// TwinCAT 3 PLC project LabExercise
// ProgramVersion: 3.1.4023.0
// libraries:
//   Tc2_NCI, * (Beckhoff Automation GmbH)
//   Tc2_Standard, * (Beckhoff Automation GmbH)
//   Tc2_System, * (Beckhoff Automation GmbH)
//   Tc3_Module, * (Beckhoff Automation GmbH)
//   VisuDialogs, * (System)
// project tree:
//   Comissioning/Function blocks/ FB_ModifyAutomaticControlSettings.TcPOU (not stored)
//   Comissioning/GVLs/ G_Commissioning.TcGVL (not stored)
//   Comissioning/Struct/ ST_AutomaticControlSettings.TcDUT (not stored), ST_ClosedLoopControlSettings.TcDUT (not stored), ST_MotionReferenceGeneratorSettings.TcDUT (not stored), ST_OpenLoopControlSettings.TcDUT (not stored)
//   ControlBox/Interfaces/ I_ControlBox.TcIO (not stored)
//   ControlBox/Function blocks/ FB_ControlBox.TcPOU (not stored), FB_RealControlBox.TcPOU (not stored), FB_VirtualControlBox.TcPOU (not stored)
//   CraneControl/Function blocks/Sub blocks/ FB_ActiveDamping.TcPOU (not stored), FB_Clock.TcPOU (not stored), FB_ClosedLoopControl.TcPOU (not stored), FB_Joystick.TcPOU (not stored), FB_MotionReferenceGenerator_limit.TcPOU (not stored), FB_OpenLoopControl.TcPOU (not stored), FB_ResetIntegralController.TcPOU (not stored), FB_Status.TcPOU (not stored)
//   CraneControl/Enums/ E_Mode.TcDUT (not stored), E_Status.TcDUT (not stored)
//   CraneControl/Function blocks/Main blocks/ FB_AutomaticControl.TcPOU (not stored), FB_ManualControl.TcPOU (not stored)
//   CraneControl/Functions/ F_BarToEng.TcPOU (not stored), F_LminToEng.TcPOU (not stored), F_RadToDeg.TcPOU (not stored)
//   CraneControl/GVLs/ G_Parameters.TcGVL (not stored), G_Work.TcGVL (not stored)
//   CraneControl/Struct/ ST_ActiveDamping.TcDUT (not stored), ST_Parameters.TcDUT (not stored)
//   / GlobalTextList.TcGTLO (not stored), PlcTask.TcTTO (not stored), Simulator.TcTTO (not stored), Visualization Manager.TcVMO (not stored)
//   HMI/ HMI.TcVIS (not stored)
//   HMI/Sub/ CommissioningHMI.TcVIS (not stored), VirtualControlBox.TcVIS (not stored)
//   Inputs/ FB_JoystickInputScaling.TcPOU (not stored), FB_PositionInputScaling.TcPOU (not stored), FB_PressureInputScaling.TcPOU (not stored), G_Inputs.TcGVL (not stored), G_Sensors.TcGVL
//   Inputs/Struct/ ST_AnalogInput.TcDUT (not stored), ST_AnalogInputStatus.TcDUT (not stored)
//   Internship/ c_FB_ControlBlockWithMonito.TcPOU, FB_Filtering.TcPOU (not stored), FB_InitialPos.TcPOU (not stored), FB_InitialPressure.TcPOU, FB_JoystickRef.TcPOU, FB_Joystick_2.TcPOU, FB_RunClock.TcPOU, FB_MotionReference.TcPOU, FB_SineMotionRef.TcPOU, G_Filtered.TcGVL (not stored), G_OPC_UA.TcGVL, G_Parameter.TcGVL, G_ControlInit.TcGVL
//   Outputs/ FB_ValveOutput.TcPOU, G_Outputs.TcGVL (not stored)
//   Outputs/Struct/ ST_pValveDeadBand.TcDUT, ST_ValveOutput.TcDUT (not stored)
//   ControlBox/GVLs/ G_VirtualControlBox.TcGVL (not stored)
//   Programs/ MAIN.TcPOU, P_ControlBlock.TcPOU, P_Commissioning.TcPOU (not stored), P_ControlBox.TcPOU (not stored), P_CraneControl.TcPOU, P_Filtering.TcPOU, P_Inputs.TcPOU, P_IntialPressure.TcPOU, P_Outputs.TcPOU (not stored), P_RunClock.TcPOU, P_Simulator.TcPOU (not stored)
//   Simulator/ FB_CraneSimulator.TcPOU (not stored), G_Simulator.TcGVL (not stored)
// real-time tasks:
//   TASK PlcTask: cycle T#1ms, priority 20, ADS port 350
//   TASK Simulator: cycle T#100us, priority 1, ADS port 351
// I/O:
//   DEVICE Device 5 (EtherCAT), AmsNetId 10.229.3.117.6.1
//     RIO (EK1100) [EK1100 EtherCAT Coupler (2A E-Bus)]
//       DI (EL1008) [EL1008 8Ch. Dig. Input 24V, 3ms]
//       DO (EL2008) [EL2008 8Ch. Dig. Output 24V, 0.5A]
//       AI1 (EL3068) [EL3068 8Ch. Ana. Input 0-10V]
//       AI2 (EL3068) [EL3068 8Ch. Ana. Input 0-10V]
//       AI3 (EL3174) [EL3174 4Ch. Ana. Input +/-10V Diff., +/-20mA SingleEnded, 16 Bit]
//       AO (EL4104) [EL4104 4Ch. Ana. Output 0-10V, 16bit]
//       End Cap (EL9011) [EL9011 End Terminal]
// variable links:
//   LabExercise/LabExercise Instance <-> Device 5 (EtherCAT)/RIO (EK1100)/AI1 (EL3068)
//     PlcTask Inputs/G_Inputs.stCylPos.nValue <-> AI Standard Channel 3/Value
//     PlcTask Inputs/G_Inputs.stCylPos.stStatus <-> AI Standard Channel 3/Status
//     PlcTask Inputs/G_Inputs.stJoyX.nValue <-> AI Standard Channel 1/Value
//     PlcTask Inputs/G_Inputs.stJoyX.stStatus <-> AI Standard Channel 1/Status
//     PlcTask Inputs/G_Inputs.stJoyY.nValue <-> AI Standard Channel 2/Value
//     PlcTask Inputs/G_Inputs.stJoyY.stStatus <-> AI Standard Channel 2/Status
//     PlcTask Inputs/G_Inputs.stSpoolPos.nValue <-> AI Standard Channel 4/Value
//     PlcTask Inputs/G_Inputs.stSpoolPos.stStatus <-> AI Standard Channel 4/Status
//   LabExercise/LabExercise Instance <-> Device 5 (EtherCAT)/RIO (EK1100)/AI2 (EL3068)
//     PlcTask Inputs/G_Inputs.stPressureCompensator.nValue <-> AI Standard Channel 3/Value
//     PlcTask Inputs/G_Inputs.stPressureCompensator.stStatus <-> AI Standard Channel 3/Status
//     PlcTask Inputs/G_Inputs.stPressureLhvSide.nValue <-> AI Standard Channel 5/Value
//     PlcTask Inputs/G_Inputs.stPressureLhvSide.stStatus <-> AI Standard Channel 5/Status
//     PlcTask Inputs/G_Inputs.stPressurePistonSide.nValue <-> AI Standard Channel 4/Value
//     PlcTask Inputs/G_Inputs.stPressurePistonSide.stStatus <-> AI Standard Channel 4/Status
//     PlcTask Inputs/G_Inputs.stPressureReturn.nValue <-> AI Standard Channel 2/Value
//     PlcTask Inputs/G_Inputs.stPressureReturn.stStatus <-> AI Standard Channel 2/Status
//     PlcTask Inputs/G_Inputs.stPressureRodSide.nValue <-> AI Standard Channel 6/Value
//     PlcTask Inputs/G_Inputs.stPressureRodSide.stStatus <-> AI Standard Channel 6/Status
//     PlcTask Inputs/G_Inputs.stPressureSupply.nValue <-> AI Standard Channel 1/Value
//     PlcTask Inputs/G_Inputs.stPressureSupply.stStatus <-> AI Standard Channel 1/Status
//   LabExercise/LabExercise Instance <-> Device 5 (EtherCAT)/RIO (EK1100)/AI3 (EL3174)
//     PlcTask Inputs/G_Inputs.stFlowReturnSide.nValue <-> AI Standard Channel 1/Value
//     PlcTask Inputs/G_Inputs.stFlowReturnSide.stStatus <-> AI Standard Channel 1/Status
//   LabExercise/LabExercise Instance <-> Device 5 (EtherCAT)/RIO (EK1100)/AO (EL4104)
//     PlcTask Outputs/G_Outputs.stValveOutput.nValveOutput <-> AO Output Channel 1/Analog output
//   LabExercise/LabExercise Instance <-> Device 5 (EtherCAT)/RIO (EK1100)/DI (EL1008)
//     PlcTask Inputs/G_Inputs.bAutoModeSelector <-> Channel 1/Input
//     PlcTask Inputs/G_Inputs.bManualModeSelector <-> Channel 2/Input
//     PlcTask Inputs/G_Inputs.bStartButton <-> Channel 3/Input
//     PlcTask Inputs/G_Inputs.bStopButton <-> Channel 4/Input
//   LabExercise/LabExercise Instance <-> Device 5 (EtherCAT)/RIO (EK1100)/DO (EL2008)
//     PlcTask Outputs/G_Outputs.bGreenLight <-> Channel 1/Output
//     PlcTask Outputs/G_Outputs.bRedLight <-> Channel 2/Output
//     PlcTask Outputs/G_Outputs.stValveOutput.bEnable <-> Channel 3/Output

// ---- Outputs/Struct/ST_pValveDeadBand.TcDUT
TYPE ST_pValveDeadBand :
STRUCT
	fPosMax	: LREAL := 29460; // Positive min value [19660..29490]
	fPosMin	: LREAL := 20800; // Positive max value [19660..29490]
	fNegMin : LREAL := 18500; // Negative max value [9830..19660]
	fNegMax	: LREAL := 9830; // Negative min value [9830..19660]
END_STRUCT
END_TYPE

// ---- Inputs/G_Sensors.TcGVL
{attribute 'qualified_only'}
VAR_GLOBAL
	fJoystickY 					: LREAL;
	fPistonPosition 			: LREAL;
	fPressureSupply				: LREAL;
	fPressureReturn 			: LREAL;
	fPressurePistonSide 		: LREAL;
	fPressureLhvSide  			: LREAL;
	fPressureRodSide 			: LREAL;
END_VAR

// ---- Internship/G_OPC_UA.TcGVL
{attribute 'qualified_only'}
VAR_GLOBAL

	// Mesurements for OPC
	fXRef : LREAL ;
	fXDotRef : LREAL;
	fXReal : LREAL ;
	
	PID_OUT : LREAL;
	Error : LREAL;
	
	fPa : LREAL ;
	fPb : LREAL ;
	fPs : LREAL ;
	
	fPaFiltered : LREAL ;
	fPbFiltered : LREAL ;
	fPsFiltered : LREAL ;
	
	fUnfilteredSignal : LREAL ;
	fFilteredSignal : LREAL ;
	
	
	fU : LREAL ;
	
	fTime : LREAL;
	
END_VAR

// ---- Internship/G_Parameter.TcGVL
{attribute 'qualified_only'}
VAR_GLOBAL
	// Motion Referance parameters
	
	fPositionSetpoint_ms : LREAL := 0.3;
	fRampTime_s : LREAL := 1;
	fMaxSpeed : LREAL := 0.1;
	fHoldPositionTime_s : LREAL := 1;
	fTimeBeforeStarting_s : LREAL := 1;
	fStartVelocity : LREAL := 0;
	
	
	// Enables
	bEnablePID : BOOL := FALSE;
	bEnableU : BOOL := FALSE;	
	bMotionSelect : BOOL := FALSE;
	fCycleTime : LREAL := 0.001;
	
	// PID-constants
	Kp : LREAL := 2.0;
	Ki : LREAL := 0.0;
	Kd : LREAL := 0.0;
	
	// Filter constants
	fPressureFilterNum :LREAL := 0.003137;
	fPressureFilterDenz : LREAL := 1.0;
	fPressureFilterDen : LREAL := -0.9969;
	fPressureFilterInit : LREAL := 0;
	
	fSignalFilterNum :LREAL := 0.09516;
	fSignalFilterDenz : LREAL := 1.0;
	fSignalFilterDen : LREAL := -0.9048;
	fSignalFilterInit : LREAL := 0;
	
END_VAR

// ---- Internship/G_ControlInit.TcGVL
VAR_GLOBAL CONSTANT
	SS_INITIALIZE: SINT := 0;
	SS_STEP: SINT := 1;
END_VAR

// ---- Internship/c_FB_ControlBlockWithMonito.TcPOU
FUNCTION_BLOCK c_FB_ControlBlockWithMonito
VAR_INPUT
	ssMethodType: SINT;
	bEnableU: BOOL;
	bEnablePID: BOOL;
	bEnableFF: BOOL;
	bEnableComp: BOOL;
	
	X_real: LREAL;
	X: LREAL;
	X_dot: LREAL;
	
	Kp: LREAL;
	Ki: LREAL;
	Kd: LREAL;
	
	Ps: LREAL;
	Pa: LREAL;
	Pb: LREAL;
	
	u_filtered: LREAL;
END_VAR
VAR_OUTPUT
	U: LREAL;
	PID_OUT: LREAL;
	Error: LREAL;
	u_unfiltered: LREAL;
END_VAR
VAR
	rtb_TSamp: LREAL;
	temp1: LREAL;
	temp2: LREAL;
	c_DiscreteTimeIntegrator_DS: LREAL;
	DiscreteTransferFcn_states: LREAL;
	UD_DSTATE: LREAL;
	u_FF: LREAL;
	Q_Const : LREAL;
END_VAR


Q_Const := G_Parameter.fQConst;

CASE ssMethodType OF
    SS_INITIALIZE: 
        (* SystemInitialize for Atomic SubSystem: '<Root>/FB_ControlBlockWithMonitoring' *)
        (* InitializeConditions for DiscreteTransferFcn: '<S2>/Discrete Transfer Fcn' *)
        DiscreteTransferFcn_states := 0.0;
        (* InitializeConditions for DiscreteIntegrator: '<S2>/Discrete-Time Integrator' *)
        c_DiscreteTimeIntegrator_DS := 0.0;
        (* InitializeConditions for UnitDelay: '<S4>/UD'
         *
         * Block description for '<S4>/UD':
         *  
         *  Store in Global RAM *)
        UD_DSTATE := 0.0;
        (* End of SystemInitialize for SubSystem: '<Root>/FB_ControlBlockWithMonitoring' *)
    SS_STEP: 
        (* Outputs for Atomic SubSystem: '<Root>/FB_ControlBlockWithMonitoring' *)
        (* Sum: '<S1>/Sum1' incorporates:
         *  Outport: '<Root>/Error' *)
        Error := X - X_real;
        (* SampleTimeMath: '<S4>/TSamp' incorporates:
         *  DiscreteTransferFcn: '<S2>/Discrete Transfer Fcn'
         *
         * About '<S4>/TSamp':
         *  y = u * K where K = 1 / ( w * Ts )
         *   *)
        rtb_TSamp := (0.0009995 * DiscreteTransferFcn_states) * 1000.0;
        (* Switch: '<S1>/Switch' incorporates:
         *  Constant: '<S1>/Constant'
         *  DiscreteIntegrator: '<S2>/Discrete-Time Integrator'
         *  Outport: '<Root>/Error'
         *  Product: '<S2>/Product'
         *  Product: '<S2>/Product1'
         *  Product: '<S2>/Product2'
         *  Sum: '<S2>/Sum1'
         *  Sum: '<S4>/Diff'
         *  UnitDelay: '<S4>/UD'
         *
         * Block description for '<S4>/Diff':
         *  
         *  Add in CPU
         *
         * Block description for '<S4>/UD':
         *  
         *  Store in Global RAM *)

        IF bEnablePID THEN 
            U := ((Kp * Error) + (Ki * c_DiscreteTimeIntegrator_DS)) + ((rtb_TSamp - UD_DSTATE) * Kd);
        ELSE 
            U := 0.0;
        END_IF;
		
		IF bEnableFF THEN 
            u_FF := u_filtered;
        ELSE 
          	u_FF := 0.0;
        END_IF;

        (* End of Switch: '<S1>/Switch' *)
        

        (* Saturate: '<S1>/Saturation1' *)

        IF U > 1.0 THEN 
            PID_OUT := 1.0;
        ELSIF U >= -1.0 THEN 
            PID_OUT := U;
        ELSE 
            PID_OUT := -1.0;
        END_IF;

        (* End of Saturate: '<S1>/Saturation1' *)
        

        (* Switch: '<S1>/Switch1' incorporates:
         *  Constant: '<S1>/Constant1'
         *  Sum: '<S1>/Sum' *)

        IF bEnableU THEN 
            U := u_FF + PID_OUT;
        ELSE 
            U := 0.0;
        END_IF;

        (* End of Switch: '<S1>/Switch1' *)
        

        (* Saturate: '<S1>/Saturation' *)

        IF U > 1.0 THEN 
            (* Outport: '<Root>/U' *)
            U := 1.0;
        ELSIF U < -1.0 THEN 
            (* Outport: '<Root>/U' *)
            U := -1.0;
        END_IF;

        (* End of Saturate: '<S1>/Saturation' *)
        

        (* MATLAB Function: '<S1>/V2Q2u' *)
        (* MATLAB Function 'FB_ControlBlockWithMonitoring/V2Q2u': '<S3>:1' *)
        (* '<S3>:1:3' phi = 0.7130; *)
        (* '<S3>:1:4' A = 33.1/100^2; *)
        (* Area *)
        (* '<S3>:1:5' BW = 0; *)
        (* deadband *)
        (* '<S3>:1:6' SpoolTravel = 7; *)
        (* Maximum Spool Travel *)
        (* '<S3>:1:7' a = (SpoolTravel-BW)/25; *)
        (* Valve Slope Characteristic [mm/(L/min)] *)
        (* '<S3>:1:8' dP_0 = 7e5; *)
        (* Pressure drop with compansator *)
        (* '<S3>:1:10' if x_dot > 0 *)
		
        IF X_dot > 0.0 THEN 
            (* '<S3>:1:11' Q = x_dot * A; *)
            (* Wanted Flow *)
            (* '<S3>:1:12' dP = (Ps-Pa)*1e5; *)
            (* '<S3>:1:13' dp_ref = abs(dP_0/dP); *)
            (* dp_ref = 1; *)
            (* '<S3>:1:15' Q_star = (Q * sqrt(dp_ref)) * 6e4; *)
            (* Referance Flow [L/min] *)
            (* '<S3>:1:16' u = (Q_star * a + BW)/SpoolTravel; *)
			IF NOT(bEnableComp) THEN
            	temp2 := ABS(700000.0 / ((Ps - Pa) * 100000.0));
			ELSE
				temp2 := 1;
			END_IF
			
            u_Unfiltered := (((SQRT(temp2) * (X_dot * 0.00331)) * 60000.0) * (7/Q_Const)) / 7.0;
            (* Control Signal [-1, 1] *)
        ELSIF X_dot < 0.0 THEN 
            (* '<S3>:1:18' elseif x_dot < 0 *)
            (* '<S3>:1:19' Q = x_dot * (A*phi); *)
            (* Wanted Flow *)
            (* '<S3>:1:20' dP = (Ps-Pb)*1e5; *)
            (* '<S3>:1:21' dp_ref = abs(dP_0/dP); *)
            (* dp_ref = 1; *)
            (* '<S3>:1:23' Q_star = (Q * sqrt(dp_ref)) * 6e4; *)
            (* Referance Flow [L/min] *)
            (* '<S3>:1:24' u = (Q_star * a - BW)/SpoolTravel; *)
			IF NOT(bEnableComp) THEN
            	temp1 := ABS(700000.0 / ((Ps - Pb) * 100000.0));
			ELSE
				temp1 := 1;
			END_IF
            u_Unfiltered := (((SQRT(temp1) * (X_dot * 0.00236003)) * 60000.0) * (7/Q_Const)) / 7.0;
            (* Control Signal [-1, 1] *)
        ELSE 
            (* '<S3>:1:26' else *)
            (* '<S3>:1:27' u = 0; *)
            u_Unfiltered := 0.0;
        END_IF;

        (* End of MATLAB Function: '<S1>/V2Q2u' *)
        

        (* Saturate: '<S1>/Saturation2' *)

        IF u_Unfiltered > 1.0 THEN 
            (* Outport: '<Root>/u_Unfiltered' *)
            u_Unfiltered := 1.0;
        ELSIF u_Unfiltered < -1.0 THEN 
            (* Outport: '<Root>/u_Unfiltered' *)
            u_Unfiltered := -1.0;
        END_IF;

        (* End of Saturate: '<S1>/Saturation2' *)
        

        (* Update for DiscreteTransferFcn: '<S2>/Discrete Transfer Fcn' incorporates:
         *  Outport: '<Root>/Error' *)
        DiscreteTransferFcn_states := Error - (-0.999 * DiscreteTransferFcn_states);
        (* u_ffpdate for DiscreteIntegrator: '<S2>/Discrete-Time Integrator' incorporates:
         *  Ou_fftport: '<Root>/Error' *)
        c_DiscreteTimeIntegrator_DS := (0.001 * Error) + c_DiscreteTimeIntegrator_DS;
        (* u_ffpdate for u_ffnitDelay: '<S4>/u_ffD'
         *
         * Block description for '<S4>/u_ffD':
         *  
         *  Store in Global RAM *)
        UD_DSTATE := rtb_TSamp;
        (* End of Ou_fftpu_ffts for Su_ffbSystem: '<Root>/FB_ControlBlockWithMonitoring' *)
END_CASE;

END_FUNCTION_BLOCK

// ---- Internship/FB_InitialPressure.TcPOU
FUNCTION_BLOCK FB_InitialPressure
VAR_INPUT
	bEnable : BOOL;
	fCurrentPressure : LREAL;
END_VAR
VAR_OUTPUT
	fInitialPressure : LREAL;
END_VAR
VAR
END_VAR

IF bEnable THEN
	fInitialPressure := fInitialPressure;
ELSE 
	fInitialPressure := fCurrentPressure;
END_IF

END_FUNCTION_BLOCK

// ---- Internship/FB_JoystickRef.TcPOU
FUNCTION_BLOCK FB_JoystickRef
VAR_INPUT
	ssMethodType: SINT;
	Joystick: LREAL;
	XRealRef: LREAL;
END_VAR
VAR_OUTPUT
	fPositionReferance_m: LREAL;
	fVelocityReferance_ms: LREAL;
END_VAR
VAR
	c_DiscreteTimeIntegrator_IC: USINT;
	c_DiscreteTimeIntegrator_DS: LREAL;
END_VAR



CASE ssMethodType OF
    SS_INITIALIZE: 
        (* SystemInitialize for Atomic SubSystem: '<Root>/FB_Joystick' *)
        (* InitializeConditions for DiscreteIntegrator: '<S1>/Discrete-Time Integrator' *)
        c_DiscreteTimeIntegrator_IC := 1;
        (* End of SystemInitialize for SubSystem: '<Root>/FB_Joystick' *)
    SS_STEP: 
        (* Outputs for Atomic SubSystem: '<Root>/FB_Joystick' *)
        (* Gain: '<S1>/Gain' *)
        fVelocityReferance_ms := G_Parameter.fMaxSpeed * Joystick;
        (* DiscreteIntegrator: '<S1>/Discrete-Time Integrator' *)

        IF c_DiscreteTimeIntegrator_IC <> 0 THEN 
            c_DiscreteTimeIntegrator_DS := XRealRef;

            IF c_DiscreteTimeIntegrator_DS > 0.45 THEN 
                c_DiscreteTimeIntegrator_DS := 0.45;
            ELSIF c_DiscreteTimeIntegrator_DS < 0.0 THEN 
                c_DiscreteTimeIntegrator_DS := 0.0;
            END_IF;

        END_IF;

        (* Outport: '<Root>/fPositionReferance_m' incorporates:
         *  DiscreteIntegrator: '<S1>/Discrete-Time Integrator' *)
        fPositionReferance_m := c_DiscreteTimeIntegrator_DS;
        (* Update for DiscreteIntegrator: '<S1>/Discrete-Time Integrator' *)
        c_DiscreteTimeIntegrator_IC := 0;
        c_DiscreteTimeIntegrator_DS := (0.2 * fVelocityReferance_ms) + c_DiscreteTimeIntegrator_DS;

        IF c_DiscreteTimeIntegrator_DS > 0.45 THEN 
            c_DiscreteTimeIntegrator_DS := 0.45;
        ELSIF c_DiscreteTimeIntegrator_DS < 0.0 THEN 
            c_DiscreteTimeIntegrator_DS := 0.0;
        END_IF;

        (* End of Update for DiscreteIntegrator: '<S1>/Discrete-Time Integrator' *)
        (* End of Outputs for SubSystem: '<Root>/FB_Joystick' *)
END_CASE;

END_FUNCTION_BLOCK

// ---- Internship/FB_Joystick_2.TcPOU
FUNCTION_BLOCK FB_Joystick_2
VAR_INPUT
	ssMethodType: SINT;
	Joystick: LREAL;
	XInital: LREAL;
END_VAR
VAR_OUTPUT
	fPositionReferance_m: LREAL;
	fVelocityReferance_ms: LREAL;
END_VAR
VAR
	c_DiscreteTimeIntegrator_IC: USINT;
	c_DiscreteTimeIntegrator_DS: LREAL;
END_VAR



CASE ssMethodType OF
    SS_INITIALIZE: 
        (* SystemInitialize for Atomic SubSystem: '<Root>/FB_Joystick' *)
        (* InitializeConditions for DiscreteIntegrator: '<S1>/Discrete-Time Integrator' *)
        c_DiscreteTimeIntegrator_IC := 1;
        (* End of SystemInitialize for SubSystem: '<Root>/FB_Joystick' *)
    SS_STEP: 
        (* Outputs for Atomic SubSystem: '<Root>/FB_Joystick' *)
        (* Gain: '<S1>/Gain' *)
        fVelocityReferance_ms := G_Parameter.fMaxSpeed * Joystick;
        (* DiscreteIntegrator: '<S1>/Discrete-Time Integrator' *)

        IF c_DiscreteTimeIntegrator_IC <> 0 THEN 
            c_DiscreteTimeIntegrator_DS := XInital;

            IF c_DiscreteTimeIntegrator_DS > 0.45 THEN 
                c_DiscreteTimeIntegrator_DS := 0.45;
            ELSIF c_DiscreteTimeIntegrator_DS < 0.0 THEN 
                c_DiscreteTimeIntegrator_DS := 0.0;
            END_IF;

        END_IF;

        (* Outport: '<Root>/fPositionReferance_m' incorporates:
         *  DiscreteIntegrator: '<S1>/Discrete-Time Integrator' *)
        fPositionReferance_m := c_DiscreteTimeIntegrator_DS;
        (* Update for DiscreteIntegrator: '<S1>/Discrete-Time Integrator' *)
        c_DiscreteTimeIntegrator_IC := 0;
        c_DiscreteTimeIntegrator_DS := (0.001 * fVelocityReferance_ms) + c_DiscreteTimeIntegrator_DS;

        IF c_DiscreteTimeIntegrator_DS > 0.45 THEN 
            c_DiscreteTimeIntegrator_DS := 0.45;
        ELSIF c_DiscreteTimeIntegrator_DS < 0.0 THEN 
            c_DiscreteTimeIntegrator_DS := 0.0;
        END_IF;

        (* End of Update for DiscreteIntegrator: '<S1>/Discrete-Time Integrator' *)
        (* End of Outputs for SubSystem: '<Root>/FB_Joystick' *)
END_CASE;

END_FUNCTION_BLOCK

// ---- Internship/FB_RunClock.TcPOU
FUNCTION_BLOCK FB_RunClock
VAR_INPUT
	bStart 		: BOOL;
	bStop 		: BOOL;
	fCycleTime  : LREAL;
END_VAR
VAR_OUTPUT
	fTime : LREAL;
END_VAR
VAR
	bOnOff : BOOL;
END_VAR

IF bStop OR (G_Work.eStatus = E_Status.Off) THEN
	bOnOff := FALSE;
	fTime := 0.0;
ELSIF bOnOff OR bStart AND (G_Work.eStatus = E_Status.Starting) THEN
	bOnOff := TRUE;
	fTime := fTime + fCycleTime;
END_IF

END_FUNCTION_BLOCK

// ---- Internship/FB_MotionReference.TcPOU
FUNCTION_BLOCK FB_MotionReference
VAR_INPUT
	fStartPosition_m: LREAL;
	fStartVelocity_m: LREAL;
	fPositionSetpoint_ms: LREAL;
	fVelocitySetpoint_m: LREAL;
	fTimeBeforeStarting_s: LREAL;
	fRampTime_s: LREAL;
	fHoldPositionTime_s: LREAL;
	fClock_s: LREAL;
	bEnable: BOOL;
END_VAR
VAR_OUTPUT
	fPositionReference_m: LREAL;
	fVelocityReference_ms: LREAL;
END_VAR
VAR
	Error: DINT;
	slopeExt: LREAL;
	slopeRetr: LREAL;
	tHold: LREAL;
	x1: LREAL;
	x4: LREAL;
	x1_tmp_tmp: LREAL;
	x4_tmp: LREAL;
	x4_tmp_tmp: LREAL;
	x4_tmp_tmp_0: LREAL;
	x1_tmp: LREAL;
END_VAR


(* Outputs for Atomic SubSystem: '<Root>/FB_MotionReferenceGenerator_nolimit' *)
(* MATLAB Function: '<S1>/WaveSignal' *)
(* MATLAB Function 'FB_MotionReferenceGenerator_nolimit/WaveSignal': '<S2>:1' *)
(* '<S2>:1:2' x_SP = x_ref - x0; *)
(* '<S2>:1:3' vs=v_ref; *)
(* '<S2>:1:4' slopeExt=v0-vs; *)
slopeExt := fStartVelocity_m - fVelocitySetpoint_m;
(* '<S2>:1:5' slopeRetr=-vs-v0; *)
slopeRetr := ( -fVelocitySetpoint_m) - fStartVelocity_m;
(* '<S2>:1:7' as = vs/tRamp; *)
(* '<S2>:1:8' s_acc=(vs^2-v0^2)/as; *)
(* '<S2>:1:10' tHold=(x_SP-s_acc)/vs; *)
tHold := ((fPositionSetpoint_ms - fStartPosition_m) - (((fVelocitySetpoint_m * fVelocitySetpoint_m) - (fStartVelocity_m * fStartVelocity_m)) / (fVelocitySetpoint_m / fRampTime_s))) / fVelocitySetpoint_m;
(* '<S2>:1:12' if tHold < 0 *)

IF tHold < 0.0 THEN 
    (* '<S2>:1:13' Error = 1; *)
    Error := 1;
ELSE 
    (* '<S2>:1:14' else *)
    (* '<S2>:1:15' Error = 0; *)
    Error := 0;
END_IF;

(* '<S2>:1:18' t1=tRamp; *)
(* '<S2>:1:19' t2=tHold; *)
(* '<S2>:1:20' t3=tRamp; *)
(* '<S2>:1:21' t4=tWait; *)
(* '<S2>:1:22' t5=t1; *)
(* '<S2>:1:23' t6=t2; *)
(* '<S2>:1:24' t7=t3; *)
(* '<S2>:1:26' x = x0; *)
(* '<S2>:1:27' x1 = x0 + v0*((t0+t1)-t0)-(slopeExt/t1)*((t0+t1)-t0)^2/2; *)
x1_tmp_tmp := fTimeBeforeStarting_s + fRampTime_s;
x4 := x1_tmp_tmp - fTimeBeforeStarting_s;
x1_tmp := slopeExt / fRampTime_s;
x1 := ((x4 * fStartVelocity_m) + fStartPosition_m) - ((x1_tmp * (x4 * x4)) / 2.0);
(* '<S2>:1:28' x2 = x1 + vs*((t0+t1+t2)-(t0+t1)); *)
(* '<S2>:1:29' x4 = x_ref - v0*((t0+t1+t2+t3+t4+t5)-(t0+t1+t2+t3+t4))+(slopeRetr/t5)*((t0+t1+t2+t3+t4+t5)-(t0+t1+t2+t3+t4))^2/2; *)
x4_tmp_tmp := x1_tmp_tmp + tHold;
x4_tmp_tmp_0 := x4_tmp_tmp + fRampTime_s;
x4_tmp := x4_tmp_tmp_0 + fHoldPositionTime_s;
x4 := (x4_tmp + fRampTime_s) - x4_tmp;
x4 := (fPositionSetpoint_ms - (x4 * fStartVelocity_m)) + (((slopeRetr / fRampTime_s) * (x4 * x4)) / 2.0);
(* '<S2>:1:30' x5 = x4-vs*((t0+t1+t2+t3+t4+t5+t6)-(t0+t1+t2+t3+t4+t5)); *)
(* '<S2>:1:32' if Error == 1 *)

IF Error = 1 THEN 
    (* '<S2>:1:33' x = x0; *)
    fPositionReference_m := fStartPosition_m;
    (* '<S2>:1:34' v = v0; *)
    fVelocityReference_ms := fStartVelocity_m;
ELSIF (fClock_s >= 0.0) AND (fClock_s < fTimeBeforeStarting_s) THEN 
    (* '<S2>:1:35' elseif t>=0 && t<t0 *)
    (* '<S2>:1:36' x = x0; *)
    fPositionReference_m := fStartPosition_m;
    (* '<S2>:1:37' v = v0; *)
    fVelocityReference_ms := fStartVelocity_m;
ELSIF (fClock_s >= fTimeBeforeStarting_s) AND (fClock_s < x1_tmp_tmp) THEN 
    (* '<S2>:1:38' elseif t>=t0 && t<(t0+t1) *)
    (* '<S2>:1:39' x = x0 + v0*(t-t0)-(slopeExt/t1)*(t-t0)^2/2; *)
    slopeExt := fClock_s - fTimeBeforeStarting_s;
    fPositionReference_m := ((slopeExt * fStartVelocity_m) + fStartPosition_m) - ((x1_tmp * (slopeExt * slopeExt)) / 2.0);
    (* '<S2>:1:40' v = v0-(slopeExt/t1)*(t-t0); *)
    fVelocityReference_ms := fStartVelocity_m - (x1_tmp * slopeExt);
ELSIF (fClock_s >= x1_tmp_tmp) AND (fClock_s < x4_tmp_tmp) THEN 
    (* '<S2>:1:41' elseif t>=(t0+t1) && t<(t0+t1+t2) *)
    (* '<S2>:1:42' x = x1 + vs*(t-(t0+t1)); *)
    fPositionReference_m := ((fClock_s - x1_tmp_tmp) * fVelocitySetpoint_m) + x1;
    (* '<S2>:1:43' v = vs; *)
    fVelocityReference_ms := fVelocitySetpoint_m;
ELSIF (fClock_s >= x4_tmp_tmp) AND (fClock_s < x4_tmp_tmp_0) THEN 
    (* '<S2>:1:44' elseif t>=(t0+t1+t2) && t<(t0+t1+t2+t3) *)
    (* '<S2>:1:45' x = x2+vs*(t-(t0+t1+t2))+(slopeExt/t3)*(t-(t0+t1+t2))^2/2; *)
    tHold := (fTimeBeforeStarting_s + fRampTime_s) + tHold;
    slopeRetr := fClock_s - tHold;
    fPositionReference_m := ((((tHold - x1_tmp_tmp) * fVelocitySetpoint_m) + x1) + (slopeRetr * fVelocitySetpoint_m)) + ((x1_tmp * (slopeRetr * slopeRetr)) / 2.0);
    (* '<S2>:1:46' v = vs+(slopeExt/t3)*(t-(t0+t1+t2)); *)
    fVelocityReference_ms := (slopeRetr * (slopeExt / fRampTime_s)) + fVelocitySetpoint_m;
ELSIF (fClock_s >= x4_tmp_tmp_0) AND (fClock_s < x4_tmp) THEN 
    (* '<S2>:1:47' elseif t>=(t0+t1+t2+t3) && t<(t0+t1+t2+t3+t4) *)
    (* '<S2>:1:48' x = x_ref; *)
    fPositionReference_m := fPositionSetpoint_ms;
    (* '<S2>:1:49' v = v0; *)
    fVelocityReference_ms := fStartVelocity_m;
ELSE 
    x1_tmp := ((x1_tmp_tmp + tHold) + fRampTime_s) + fHoldPositionTime_s;
    slopeExt := x1_tmp + fRampTime_s;

    IF (fClock_s >= x1_tmp) AND (fClock_s < slopeExt) THEN 
        (* '<S2>:1:50' elseif t>=(t0+t1+t2+t3+t4) && t<(t0+t1+t2+t3+t4+t5) *)
        (* '<S2>:1:51' x = x_ref - v0*(t-(t0+t1+t2+t3+t4))+(slopeRetr/t5)*(t-(t0+t1+t2+t3+t4))^2/2; *)
        tHold := fClock_s - x1_tmp;
        slopeRetr := slopeRetr / fRampTime_s;
        fPositionReference_m := (fPositionSetpoint_ms - (tHold * fStartVelocity_m)) + ((slopeRetr * (tHold * tHold)) / 2.0);
        (* '<S2>:1:52' v = v0+(slopeRetr/t5)*(t-(t0+t1+t2+t3+t4)); *)
        fVelocityReference_ms := (tHold * slopeRetr) + fStartVelocity_m;
    ELSE 
        x1_tmp := slopeExt + tHold;

        IF (fClock_s >= slopeExt) AND (fClock_s < x1_tmp) THEN 
            (* '<S2>:1:53' elseif t>=(t0+t1+t2+t3+t4+t5) && t<(t0+t1+t2+t3+t4+t5+t6) *)
            (* '<S2>:1:54' x = x4-vs*(t-(t0+t1+t2+t3+t4+t5)); *)
            fPositionReference_m := x4 - ((fClock_s - slopeExt) * fVelocitySetpoint_m);
            (* '<S2>:1:55' v = -vs; *)
            fVelocityReference_ms :=  -fVelocitySetpoint_m;
        ELSIF (fClock_s >= x1_tmp) AND (fClock_s < (x1_tmp + fRampTime_s)) THEN 
            (* '<S2>:1:56' elseif t>=(t0+t1+t2+t3+t4+t5+t6) && t<(t0+t1+t2+t3+t4+t5+t6+t7) *)
            (* '<S2>:1:57' x = x5-vs*(t-(t0+t1+t2+t3+t4+t5+t6))-(slopeRetr/t3)*(t-(t0+t1+t2+t3+t4+t5+t6))^2/2; *)
            tHold := fClock_s - x1_tmp;
            slopeRetr := slopeRetr / fRampTime_s;
            fPositionReference_m := ((x4 - ((x1_tmp - slopeExt) * fVelocitySetpoint_m)) - (tHold * fVelocitySetpoint_m)) - ((slopeRetr * (tHold * tHold)) / 2.0);
            (* '<S2>:1:58' v = -vs-(slopeRetr/t3)*(t-(t0+t1+t2+t3+t4+t5+t6)); *)
            fVelocityReference_ms := ( -fVelocitySetpoint_m) - (tHold * slopeRetr);
        ELSE 
            (* '<S2>:1:59' else *)
            (* '<S2>:1:60' x = x0; *)
            fPositionReference_m := fStartPosition_m;
            (* '<S2>:1:61' v = v0; *)
            fVelocityReference_ms := fStartVelocity_m;
        END_IF;

    END_IF;

END_IF;

(* End of MATLAB Function: '<S1>/WaveSignal' *)


(* Switch: '<S1>/Switch' incorporates:
 *  Switch: '<S1>/Switch1' *)
(* '<S2>:1:64' T = t0+t1+t2+t3+t4+t5+t6+t7; *)

IF  NOT bEnable THEN 
    (* Outport: '<Root>/fVelocityReference_ms' *)
    fVelocityReference_ms := fStartVelocity_m;
    (* Outport: '<Root>/fPositionReference_m' *)
    fPositionReference_m := fStartPosition_m;
END_IF;

(* End of Switch: '<S1>/Switch' *)
(* End of Outputs for SubSystem: '<Root>/FB_MotionReferenceGenerator_nolimit' *)

END_FUNCTION_BLOCK

// ---- Internship/FB_SineMotionRef.TcPOU
FUNCTION_BLOCK FB_SineMotionRef
VAR_INPUT
	ssMethodType: SINT;
	fTime: LREAL;
	fPos_Ramp_Time: LREAL;
	fPeak_pos: LREAL;
	fStart_vel: LREAL;
	fStart_time: LREAL;
	fHold_time: LREAL;
	fXReal: LREAL;
END_VAR
VAR_OUTPUT
	X_dot: LREAL;
	X: LREAL;
END_VAR
VAR
	peak_vel: LREAL;
	amplitude_vel: LREAL;
	c_DiscreteTimeIntegrator_DS: LREAL;
END_VAR



CASE ssMethodType OF
    SS_INITIALIZE: 
        (* SystemInitialize for Atomic SubSystem: '<Root>/FB_SineMotionRef' *)
        (* InitializeConditions for DiscreteIntegrator: '<S1>/Discrete-Time Integrator' *)
        c_DiscreteTimeIntegrator_DS := 0.0;
        (* End of SystemInitialize for SubSystem: '<Root>/FB_SineMotionRef' *)
    SS_STEP: 
        (* Outputs for Atomic SubSystem: '<Root>/FB_SineMotionRef' *)
        (* MATLAB Function: '<S1>/MATLAB Function' *)
        (* MATLAB Function 'FB_SineMotionRef/MATLAB Function': '<S2>:1' *)
        (* '<S2>:1:2' max_pos = peak_pos-start_pos; *)
        (* '<S2>:1:3' peak_vel = max_pos*2/pos_ramp_time; *)
        peak_vel := ((fPeak_pos - fXReal) * 2.0) / fPos_Ramp_Time;
        (* '<S2>:1:4' pos_sat = peak_vel*pos_ramp_time/2 +start_pos; *)
        (* '<S2>:1:5' amplitude_vel = peak_vel/2; *)
        amplitude_vel := peak_vel / 2.0;
        (* '<S2>:1:6' if pos_sat <= 0.4 *)

        IF (((peak_vel * fPos_Ramp_Time) / 2.0) + fXReal) <= 0.4 THEN 
            (* '<S2>:1:7' if time<start_time *)

            IF fTime < fStart_time THEN 
                (* '<S2>:1:8' X_dot=start_vel; *)
                X_dot := fStart_vel;
            ELSIF fTime <= (fPos_Ramp_Time + fStart_time) THEN 
                (* '<S2>:1:9' elseif time<=pos_ramp_time+start_time *)
                (* '<S2>:1:10' X_dot=amplitude_vel-amplitude_vel*cos((2*(time-start_time))/pos_ramp_time*pi)+start_vel; *)
                X_dot := (amplitude_vel - (COS((((fTime - fStart_time) * 2.0) / fPos_Ramp_Time) * 3.1415926535897931) * amplitude_vel)) + fStart_vel;
            ELSIF fTime < ((fHold_time + fPos_Ramp_Time) + fStart_time) THEN 
                (* '<S2>:1:11' elseif time<hold_time+pos_ramp_time+start_time *)
                (* '<S2>:1:12' X_dot=start_vel; *)
                X_dot := fStart_vel;
            ELSIF fTime < (((2.0 * fPos_Ramp_Time) + fHold_time) + fStart_time) THEN 
                (* '<S2>:1:13' elseif time< hold_time+2*pos_ramp_time+start_time *)
                (* '<S2>:1:14' X_dot=-(amplitude_vel-amplitude_vel*cos((2*(time-(start_time +hold_time+pos_ramp_time)))/pos_ramp_time*pi)+start_vel); *)
                X_dot :=  -((amplitude_vel - (COS((((fTime - ((fStart_time + fHold_time) + fPos_Ramp_Time)) * 2.0) / fPos_Ramp_Time) * 3.1415926535897931) * amplitude_vel)) + fStart_vel);
            ELSE 
                (* '<S2>:1:15' else *)
                (* '<S2>:1:16' X_dot=start_vel; *)
                X_dot := fStart_vel;
            END_IF;

        ELSE 
            (* '<S2>:1:18' else *)
            (* '<S2>:1:19' X_dot=0; *)
            X_dot := 0.0;
        END_IF;

        (* End of MATLAB Function: '<S1>/MATLAB Function' *)
        

        (* Outport: '<Root>/X' incorporates:
         *  DiscreteIntegrator: '<S1>/Discrete-Time Integrator'
         *  Sum: '<S1>/Sum' *)
        X := c_DiscreteTimeIntegrator_DS + fXReal;
        (* Update for DiscreteIntegrator: '<S1>/Discrete-Time Integrator' *)
        c_DiscreteTimeIntegrator_DS := (0.001 * X_dot) + c_DiscreteTimeIntegrator_DS;
        (* End of Outputs for SubSystem: '<Root>/FB_SineMotionRef' *)
END_CASE;

END_FUNCTION_BLOCK

// ---- Outputs/FB_ValveOutput.TcPOU
FUNCTION_BLOCK FB_ValveOutput
VAR_INPUT
	bEnable 			: BOOL;
	stParam 			: ST_Parameters;
	fNormalizedInput 	: LREAL;
END_VAR
VAR_OUTPUT
	bEnableValveOutput : BOOL;
	nOutput : INT; 
END_VAR
VAR
	nOffset 	: INT := 19630;
	nMaxValue	: INT := 29460;
	nMinValue 	: INT :=  9830;
	nTempOutput : INT;
END_VAR

IF fNormalizedInput > 0.0 THEN
	nTempOutput := LREAL_TO_INT(ABS(fNormalizedInput*(stParam.stValveDeadBand.fPosMax - stParam.stValveDeadBand.fPosMin) + stParam.stValveDeadBand.fPosMin));
ELSIF fNormalizedInput < 0.0 THEN
	nTempOutput := LREAL_TO_INT(ABS(fNormalizedInput*(stParam.stValveDeadBand.fNegMax - stParam.stValveDeadBand.fNegMin) - stParam.stValveDeadBand.fNegMin));
ELSE
	nTempOutput := nOffset;
END_IF

IF NOT(bEnable) THEN
	nOutput := nOffset;
	bEnableValveOutput := FALSE;
ELSE
	nOutput := LIMIT(nMinValue, nTempOutput, nMaxValue);
	bEnableValveOutput := TRUE; 
END_IF

END_FUNCTION_BLOCK

// ---- Programs/MAIN.TcPOU
PROGRAM MAIN
VAR
END_VAR

P_Commissioning();
P_ControlBox();
P_Filtering();
P_CraneControl();
P_ControlBlock();
P_Outputs();
P_Inputs();
P_RunClock();

END_PROGRAM

// ---- Programs/P_Filtering.TcPOU
PROGRAM P_Filtering
VAR
	fbControlBlock : c_FB_ControlBlockWithMonito;
	fbFilterPa : FB_Filtering;
	fbFilterPb : FB_Filtering;
	fbFilterPs : FB_Filtering;
	fbFilterU : FB_Filtering;
END_VAR

fbFilterPa(
	ssMethodType := 1,
	Signal := G_Sensors.fPressurePistonSide,
	Num := G_Parameter.fPressureFilterNum,
	Denz := G_Parameter.fPressureFilterDenz,
	Den := G_Parameter.fPressureFilterDen,
	Initial := G_Parameter.fPressureFilterInit,
	
	Signal_Filtered => G_Filtered.fPressurePistonSideFiltered,
	Signal_Filtered => G_OPC_UA.fPaFiltered
);

fbFilterPb(
	ssMethodType := 1,
	Signal := G_Sensors.fPressureRodSide,
	Num := G_Parameter.fPressureFilterNum,
	Denz := G_Parameter.fPressureFilterDenz,
	Den := G_Parameter.fPressureFilterDen,
	Initial := G_Parameter.fPressureFilterInit,
	
	Signal_Filtered => G_Filtered.fPressureRodSideFiltered,
	Signal_Filtered => G_OPC_UA.fPbFiltered
);

fbFilterPs(
	ssMethodType := 1,
	Signal := G_Sensors.fPressureSupply,
	Num := G_Parameter.fPressureFilterNum,
	Denz := G_Parameter.fPressureFilterDenz,
	Den := G_Parameter.fPressureFilterDen,
	Initial := G_Parameter.fPressureFilterInit,
	
	Signal_Filtered => G_Filtered.fPressureSupplyFiltered,
	Signal_Filtered => G_OPC_UA.fPsFiltered
);

fbFilterU(
	ssMethodType := 1,
	Signal := G_Filtered.fValveOutputUnfiltered,
	Num := G_Parameter.fSignalFilterNum,
	Denz := G_Parameter.fSignalFilterDenz,
	Den := G_Parameter.fSignalFilterDen,
	Initial := G_Parameter.fSignalFilterInit,
	
	Signal_Filtered => G_Filtered.fValveOutputFiltered,
	Signal_Filtered => G_OPC_UA.fFilteredSignal
);

END_PROGRAM

// ---- Programs/P_CraneControl.TcPOU
PROGRAM P_CraneControl
VAR
 	fbStatus 					: FB_Status;
	fbRunningClock 				: FB_Clock;
	fbManualControl 			: FB_ManualControl; 
	bEnableManualControl 		: BOOL;
	fbAutomaticControl 			: FB_AutomaticControl;
	bEnableAutomaticControl 	: BOOL; 
	fbActiveDamping 			: FB_ActiveDamping;
	fControlOutputNormalized 	: LREAL; 
	
	ADtest0 : LREAL;
	ADtest1 : LREAL;
	ADtest2 : LREAL;
	ADtest : BOOL;
END_VAR

fbStatus(
bFault := G_Work.bFault,
eMode := G_Work.eMode,
fTime := fbRunningClock.fTime,
eStatus => G_Work.eStatus
);

fbRunningClock(
	bStart := (fbStatus.eStatus = E_Status.Starting) OR (fbStatus.eStatus = E_Status.Running),
	bStop := (fbStatus.eStatus = E_Status.Stopping),
	fCycleTime := G_Parameters.stParam.fCyclicTime
);


fbManualControl(
	eMode := G_Work.eMode,
	eStatus := G_Work.eStatus,
	stParam := G_Parameters.stParam, 
);

fbAutomaticControl(
	eMode := G_Work.eMode,
	eStatus := G_Work.eStatus,
	stAutomaticControlSettings := G_Commissioning.stAutomaticControlSettings,
	stMotionReferenceGeneratorSettings := G_Commissioning.stMotionReferenceGeneratorSettings,
	stParam := G_Parameters.stParam,
	fPositionFeedback := G_Sensors.fPistonPosition
);

fbActiveDamping(
	ssMethodType := BOOL_TO_SINT(G_Commissioning.stAutomaticControlSettings.bEnableActiveDamping),
	bEnable := (fbStatus.eStatus = E_Status.Running),
	stParam := G_Parameters.stParam,
	fPressurePistonSide_Pa := F_BarToEng(G_Sensors.fPressurePistonSide),
	fPressureRodSide_Pa := F_BarToEng(G_Sensors.fPressureRodSide)
);

IF (G_Work.eMode = E_Mode.Manual AND G_Work.eStatus = E_Status.Running) THEN
	fControlOutputNormalized := LIMIT(-1.0, (fbManualControl.fControlOutputNormalized - fbActiveDamping.fPressureFeedbackNormalized), 1.0);
ELSIF (G_Work.eMode = E_Mode.Auto AND G_Work.eStatus = E_Status.Running) THEN
	fControlOutputNormalized := LIMIT(-1.0, (-fbAutomaticControl.fControlOutputNormalized - fbActiveDamping.fPressureFeedbackNormalized), 1.0);
ELSE
	fControlOutputNormalized := 0.0;
END_IF

//G_Work.fControlOutputNormalized := fControlOutputNormalized;

END_PROGRAM

// ---- Programs/P_ControlBlock.TcPOU
PROGRAM P_ControlBlock
VAR
	fbControlBlock : c_FB_ControlBlockWithMonito;
	fbMotionRef : FB_MotionReference;
	fbSineMotionRef : FB_SineMotionRef;
	fbJoyRef : FB_Joystick_2;
	fbClock : FB_Clock;
	fbInitialPos : FB_InitialPos;	
END_VAR

fbClock(
	bStart := G_Inputs.bStartButton,
	bStop := G_Inputs.bStopButton,
	fCycleTime :=0.001
);

fbInitialPos(
	bEnable := (G_Work.eStatus = E_Status.Running),
	fCurrentPos := G_Sensors.fPistonPosition,
);

IF (G_Work.eMode = E_Mode.Auto) THEN
	
	G_OPC_UA.fXRef := fbMotionRef.fPositionReference_m;
	G_OPC_UA.fXDotRef := fbMotionRef.fVelocityReference_ms;
	
	IF (G_Parameter.bMotionSelect) THEN
		fbMotionRef(
			fStartPosition_m := fbInitialPos.fInitialPos,
			fStartVelocity_m := G_Parameter.fStartVelocity,
			fPositionSetpoint_ms := G_Parameter.fPositionSetpoint_ms,
			fVelocitySetpoint_m := G_Parameter.fMaxSpeed,
			fTimeBeforeStarting_s := G_Parameter.fTimeBeforeStarting_s,
			fRampTime_s := G_Parameter.fRampTime_s,
			fHoldPositionTime_s := G_Parameter.fHoldPositionTime_s,
			fClock_s:= fbClock.fTime,
			bEnable:= G_Inputs.bStartButton		
		);
		
		fbControlBlock(
		ssMethodType := BOOL_TO_SINT(G_Work.eStatus = E_Status.Running),

		X_dot := fbMotionRef.fVelocityReference_ms,
		X := fbMotionRef.fPositionReference_m,

	);
	ELSE
		fbSineMotionRef(
			ssMethodType := BOOL_TO_SINT(G_Work.eStatus = E_Status.Running),
			fTime := fbClock.fTime,
			fPos_Ramp_Time := G_Parameter.fRampTime_s,
			fPeak_pos := G_Parameter.fPositionSetpoint_ms,
			fStart_vel := G_Parameter.fStartVelocity,
			fStart_time := G_Parameter.fTimeBeforeStarting_s,
			fHold_time := G_Parameter.fHoldPositionTime_s,
			fXReal := G_Sensors.fPistonPosition 
		);
		
		fbControlBlock(
			ssMethodType := BOOL_TO_SINT(G_Work.eStatus = E_Status.Running),

			X_dot := fbSineMotionRef.X_dot,
			X := fbSineMotionRef.X,

		);
	END_IF
			fbControlBlock(
			ssMethodType := BOOL_TO_SINT(G_Work.eStatus = E_Status.Running),
			bEnablePID := G_Parameter.bEnablePID,
			bEnableU := G_Parameter.bEnableU,
		
			X_real:= G_Sensors.fPistonPosition,
		
			Kp := G_Parameter.Kp,
			Ki := G_Parameter.Ki,
			Kd := G_Parameter.Kd,
		
			Pa:= G_Filtered.fPressurePistonSideFiltered, 
			Pb := G_Filtered.fPressureRodSideFiltered,
			Ps:= G_Filtered.fPressureSupplyFiltered,
		
			u_filtered := G_Filtered.fValveOutputFiltered,
		
			u_Unfiltered => G_Filtered.fValveOutputUnfiltered,
			u_Unfiltered => G_OPC_UA.fUnfilteredSignal,
		
			U	=> G_Work.fControlOutputNormalized,
			U	=> G_OPC_UA.fU,
		
			Error => G_OPC_UA.Error
		);

ELSIF (G_Work.eMode = E_Mode.Manual) THEN

	G_OPC_UA.fXRef := fbJoyRef.fPositionReferance_m;
	G_OPC_UA.fXDotRef := fbJoyRef.fVelocityReferance_ms;
	
	fbJoyRef(
		ssMethodType := BOOL_TO_SINT(G_Work.eStatus = E_Status.Running),
		Joystick := G_Sensors.fJoystickY,
		XInital := fbInitialPos.fInitialPos,
	);

	
	fbControlBlock(
	ssMethodType := BOOL_TO_SINT(G_Work.eStatus = E_Status.Running),
	bEnablePID := G_Parameter.bEnablePID,
	bEnableU := G_Parameter.bEnableU,
		
	X_real:= G_Sensors.fPistonPosition,
	X_dot := fbJoyRef.fVelocityReferance_ms,
	X := fbJoyRef.fPositionReferance_m,
	
	Kp := G_Parameter.Kp,
	Ki := G_Parameter.Ki,
	Kd := G_Parameter.Kd,
	
	Pa:= G_Filtered.fPressurePistonSideFiltered, 
	Pb := G_Filtered.fPressureRodSideFiltered,
	Ps:= G_Filtered.fPressureSupplyFiltered,
	
	u_filtered := G_Filtered.fValveOutputFiltered,
		
	u_Unfiltered => G_Filtered.fValveOutputUnfiltered,
	u_Unfiltered => G_OPC_UA.fUnfilteredSignal,
	
	U	=> G_Work.fControlOutputNormalized,
	U	=> G_OPC_UA.fU,
	
	Error => G_OPC_UA.Error
	);
END_IF

END_PROGRAM

// ---- Programs/P_Inputs.TcPOU
PROGRAM P_Inputs
VAR
	fbJoystick 				: FB_JoystickInputScaling;
	fbPositionSensor 		: FB_PositionInputScaling;
	fbPressureSupplySensor 	: FB_PressureInputScaling;
	fbPressureReturnSensor 	: FB_PressureInputScaling;
	fbPressurePistonSide 	: FB_PressureInputScaling;
	fbPressureLhvSide 		: FB_PressureInputScaling;
	fbPressureRodSide 		: FB_PressureInputScaling;
END_VAR

fbJoystick(
	bEnable := G_Inputs.bManualModeSelector,
	nRawInput := G_Inputs.stJoyY.nValue,
	fOutput => G_Sensors.fJoystickY
);

fbPositionSensor(
	nRawInput := G_Inputs.stCylPos.nValue,
	fOutput => G_Sensors.fPistonPosition,
	fOutput => G_OPC_UA.fXReal
);

fbPressureSupplySensor(
	nRawInput := G_Inputs.stPressureSupply.nValue,
	fOutput => G_Sensors.fPressureSupply,
	fOutput => G_OPC_UA.fPs
);

fbPressureReturnSensor(
	nRawInput := G_Inputs.stPressureReturn.nValue,
	fOutput => G_Sensors.fPressureReturn
);

fbPressurePistonSide(
	nRawInput := G_Inputs.stPressurePistonSide.nValue,
	fOutput => G_Sensors.fPressurePistonSide,
	fOutput => G_OPC_UA.fPa
);

fbPressureLhvSide(
	nRawInput := G_Inputs.stPressureLhvSide.nValue,
	fOutput => G_Sensors.fPressureLhvSide
);

fbPressureRodSide(
	nRawInput := G_Inputs.stPressureRodSide.nValue,
	fOutput => G_Sensors.fPressureRodSide,
	fOutput => G_OPC_UA.fPb
);

END_PROGRAM

// ---- Programs/P_RunClock.TcPOU
PROGRAM P_RunClock
VAR
	fbRunClock : FB_RunClock;
END_VAR

fbRunClock(
	bStart := TRUE,
	bStop := G_Inputs.bStopButton,
	fCycleTime := G_Parameter.fCycleTime,
	
	fTime => G_OPC_UA.fTime
);

END_PROGRAM

// ---- Programs/P_IntialPressure.TcPOU
PROGRAM P_IntialPressure
VAR
END_VAR

END_PROGRAM
